// TIA Portal V18 export
// export: Created 2026-06-08T17:01:57.7650911Z, ExportSetting WithDefaults, DisplayName Totally Integrated Automation Portal, DisplayVersion V18, DisplayName TIA Portal Openness, DisplayVersion V18, DisplayName TIA Portal Version Control Interface, DisplayVersion V18, DisplayName STEP 7 Professional, DisplayVersion V18, DisplayName STEP 7 Safety, DisplayVersion V18, DisplayName WinCC Professional, DisplayVersion V18
VAR_GLOBAL   // PLC tag table "Default tag table"
   PB_MAIN_MOVE_R AT %I0.0 : Bool;
   PB_MAIN_MOVE_F AT %I0.1 : Bool;
   PB_MAIN_STOP AT %I0.2 : Bool;
   SENSOR_HOME AT %I0.3 : Bool;
   SENSOR_FINISH_1 AT %I0.4 : Bool;
   PB_EMERGENCY AT %I0.5 : Bool;
   PB_RESET AT %I0.6 : Bool;
   MAIN_COIL_R AT %Q0.0 : Bool;
   MAIN_COIL_F AT %Q0.1 : Bool;
   COIL_EMERGENCY AT %Q0.2 : Bool;
   System_Byte AT %MB1 : Byte;
   FirstScan AT %M1.0 : Bool;
   DiagStatusUpdate AT %M1.1 : Bool;
   AlwaysTRUE AT %M1.2 : Bool;
   AlwaysFALSE AT %M1.3 : Bool;
   Clock_Byte AT %MB0 : Byte;
   Clock_10Hz AT %M0.0 : Bool;
   Clock_5Hz AT %M0.1 : Bool;
   "Clock_2.5Hz" AT %M0.2 : Bool;
   Clock_2Hz AT %M0.3 : Bool;
   "Clock_1.25Hz" AT %M0.4 : Bool;
   Clock_1Hz AT %M0.5 : Bool;
   "Clock_0.625Hz" AT %M0.6 : Bool;
   "Clock_0.5Hz" AT %M0.7 : Bool;
   M1_RESET_COUNT AT %I0.7 : Bool;
   PB_M1_MOVE_R AT %I1.0 : Bool;
   PB_M1_MOVE_F AT %I1.1 : Bool;
   PB_M1_STOP AT %I1.2 : Bool;
   M1_COIL_R AT %Q0.3 : Bool;
   M1_COIL_F AT %Q0.4 : Bool;
   SENSOR_FINISH_2 AT %I1.3 : Bool;
   M2_RESET_COUNTER AT %I1.4 : Bool;
   PB_M2_MOVE_R AT %I1.5 : Bool;
   M2_COIL_R AT %Q0.5 : Bool;
   M2_COIL_F AT %Q0.6 : Bool;
   PB_M2_MOVE_F AT %I8.0 : Bool;
   PB_M2_STOP AT %I8.1 : Bool;
   DIVIDER_1 AT %Q8.0 : Bool;
   DIVIDER_2 AT %Q8.1 : Bool;
END_VAR
